TYPE ST_BagOpen :
STRUCT
	bag_status				: BagStatus;
	iCnt_sensor_detection	: INT;
	sensor_status			: STRING;
END_STRUCT
END_TYPE

(* stored: Version 1.1.0.1, ProductVersion 3.1.4024.12
   DUT ST_BagOpen: Id {99f9e337-7847-4d36-8e88-ee012a1dcec5} *)
